// TwinCAT 3 PLC project MAS418_PLC
// ProgramVersion: 3.1.4023.0
// libraries:
//   Tc2_Standard, * (Beckhoff Automation GmbH)
//   Tc2_System, * (Beckhoff Automation GmbH)
//   Tc3_Module, * (Beckhoff Automation GmbH)
//   VisuDialogs, * (System)
// project tree:
//   / GlobalTextList.TcGTLO, PlcTask.TcTTO, Visualization Manager.TcVMO (not stored)
//   POUs/ MAIN.TcPOU
//   VISUs/ HMI.TcVIS
// real-time tasks:
//   TASK PlcTask: cycle T#10ms, priority 20, ADS port 350

CONFIGURATION MAS418_PLC
    RESOURCE PLC ON TwinCAT3
        TASK PlcTask(INTERVAL := T#10ms, PRIORITY := 20);
        PROGRAM MAIN WITH PlcTask : MAIN;
    END_RESOURCE
END_CONFIGURATION

// ---- POUs/MAIN.TcPOU
PROGRAM MAIN
VAR
	bEnable : BOOL;
	bStart: BOOL;
	nINT: INT:= -32768;
	nUINT: UINT:= 65535;
	fREAL: REAL:= 255.255;
	sPowerStatus : STRING:= 'Power Off';
END_VAR

bEnable := bStart;

END_PROGRAM

// ---- GlobalTextList.TcGTLO
TEXTLIST GlobalTextList
  415 = '%f'
  726 = '%i'
  548 = '%s'
  7 = 'BOOL'
  893 = 'DataTypeTesting'
  57 = 'helo'
  484 = 'INT'
  862 = 'Power ON'
  612 = 'REAL'
  853 = 'STRING'
  25 = 'UINT'
END_TEXTLIST

// ---- VISUs/HMI.TcVIS
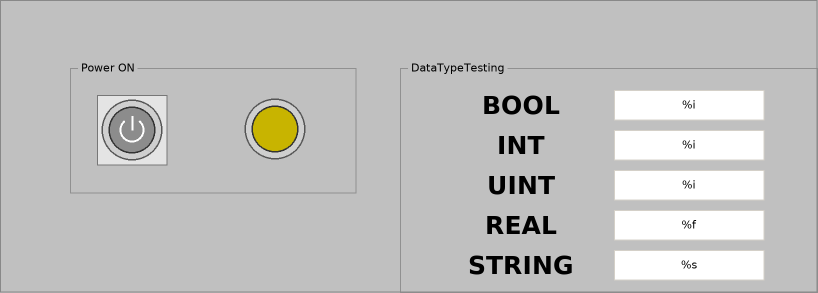
VISUALIZATION HMI  // 818x293
    GroupBox (400,60 418x233), "DataTypeTesting"
        Textfield (214,30 150x30), "%i", text variable: MAIN.bEnable
        Label (46,30 150x30), "BOOL"
        Textfield (214,70 150x30), "%i", text variable: MAIN.nINT
        Label (46,70 150x30), "INT"
        Textfield (214,110 150x30), "%i", text variable: MAIN.nUINT
        Label (46,110 150x30), "UINT"
        Textfield (214,150 150x30), "%f", text variable: MAIN.fREAL
            OnMouseDown: write the text variable via Default
        Label (46,150 150x30), "REAL"
        Textfield (214,190 150x30), "%s", text variable: MAIN.sPowerStatus
            OnMouseDown: write the text variable via Default
        Label (46,190 150x30), "STRING"
    GroupBox (70,60 286x133), "Power ON"
        PowerSwitch (27,35 70x70), variable: MAIN.bStart, behaviour: TOGGLE, style: Switch-PowerSwitch-Gray
        Lamp1 (170,34 70x70), variable: MAIN.bEnable, style: Lamp-Lamp1-Yellow
END_VISUALIZATION
